// LS Electric XG5000 project: 485모드
// PLC LSPLC

PROGRAM NewProgram (task: 스캔 프로그램)

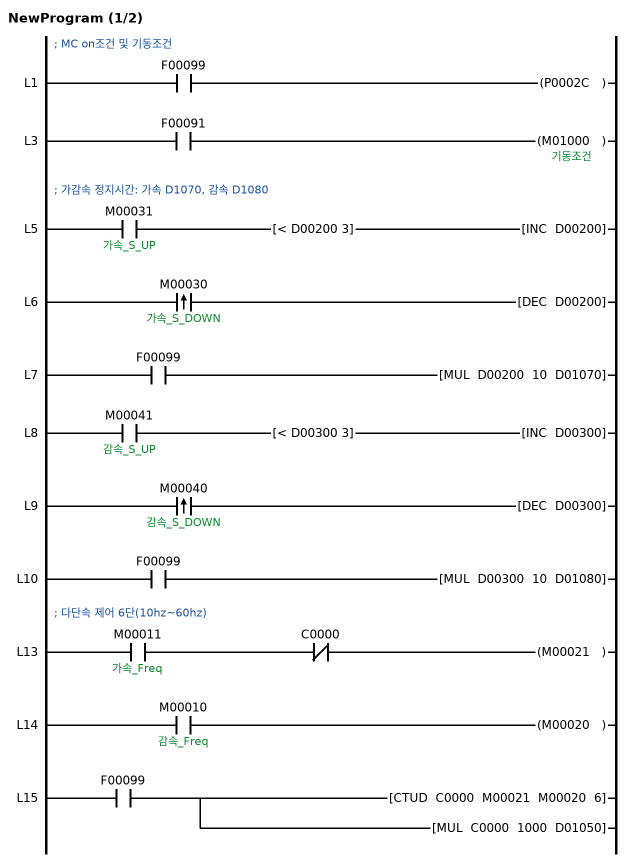
// MC on조건 및 기동조건
; L1
LOAD      F00099
OUT       P0002C
; L3
LOAD      F00091
OUT       M01000	// 기동조건
// 가감속 정지시간: 가속 D1070, 감속 D1080
; L5
LOAD      M00031	// 가속_S_UP
AND<      D00200 3
INC       D00200
; L6
LOADP     M00030	// 가속_S_DOWN
DEC       D00200
; L7
LOAD      F00099
MUL       D00200 10 D01070
; L8
LOAD      M00041	// 감속_S_UP
AND<      D00300 3
INC       D00300
; L9
LOADP     M00040	// 감속_S_DOWN
DEC       D00300
; L10
LOAD      F00099
MUL       D00300 10 D01080
// 다단속 제어 6단(10hz~60hz)
; L13
LOAD      M00011	// 가속_Freq
AND NOT   C0000
OUT       M00021
; L14
LOAD      M00010	// 감속_Freq
OUT       M00020
; L15
LOAD      F00099
CTUD      C0000 M00021 M00020 6
MUL       C0000 1000 D01050

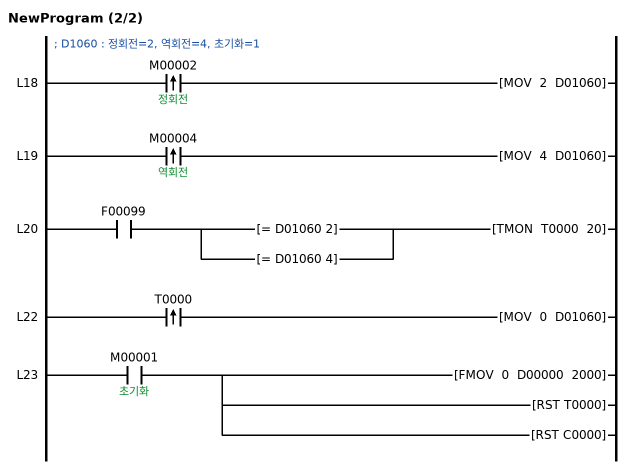
// D1060 : 정회전=2, 역회전=4, 초기화=1
; L18
LOADP     M00002	// 정회전
MOV       2 D01060
; L19
LOADP     M00004	// 역회전
MOV       4 D01060
; L20
LOAD      F00099
LOAD=     D01060 2
OR=       D01060 4
AND LOAD
TMON      T0000 20
; L22
LOADP     T0000
MOV       0 D01060
; L23
LOAD      M00001	// 초기화
FMOV      0 D00000 2000
RST       T0000
RST       C0000